TYPE ST_HeightLimits :
STRUCT
	
	nHigh					: REAL;
	nLow					: REAL;

END_STRUCT
END_TYPE

(* stored: Version 1.1.0.1, ProductVersion 3.1.4024.13
   DUT ST_HeightLimits: Id {a1184038-8f28-4448-b113-60f68d8d1719} *)
